Staubli VAL3: delete.pgx

public program delete(string x_sName, num& x_nResult[])
  local string l_sItem
  local num l_nSize
begin
  //
  // delete the select trajectory
  //
end
